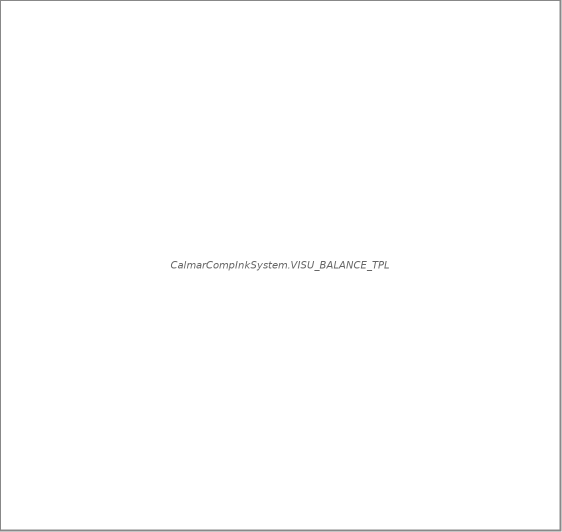
VISUALIZATION VISU_BALANCE  // 562x532
    Frame (0,0 560x530)
        shows CalmarCompInkSystem.VISU_BALANCE_TPL(m_Idx_Max := CONFIGURATION.iCIk_NB_INKBALANCE, m_ModId_StAdsStorageTank := PRG_INK.sAdsIkInkStorageTank[PRG_INK.iL_SelectedBalance], m_ModId_FbBalanceMonitor := PRG_INK.FB_Balance[PRG_INK.iL_SelectedBalance], m_Idx := PRG_INK.iL_SelectedBalance)
END_VISUALIZATION

(* stored: Version 1.1.0.1, ProductVersion 3.1.4024.9
   Visu VISU_BALANCE: Id {2ef4fb25-255a-4ca0-a053-813df686fb2c} *)
